DATA_BLOCK "dbArchiveSlotTank"
{ S7_Optimized_Access := 'TRUE' }
VERSION : 0.8
NON_RETAIN
"fbArchiveSlotTank"

BEGIN

END_DATA_BLOCK

